// TIA Portal V19 export
FUNCTION "FC30_DoorAcces" : Void   // FC30, LAD
{ S7_Optimized_Access := 'TRUE' }
// stored: AutoNumber false, IsIECCheckEnabled true, SetENOAutomatically false
   VAR_TEMP
      xt_RobotStopped : Bool;
      xt_Robot1Stopped : Bool;
      xt_Robot2Stopped : Bool;
   END_VAR
BEGIN

REGION Network 1: Robot 1 is stopped
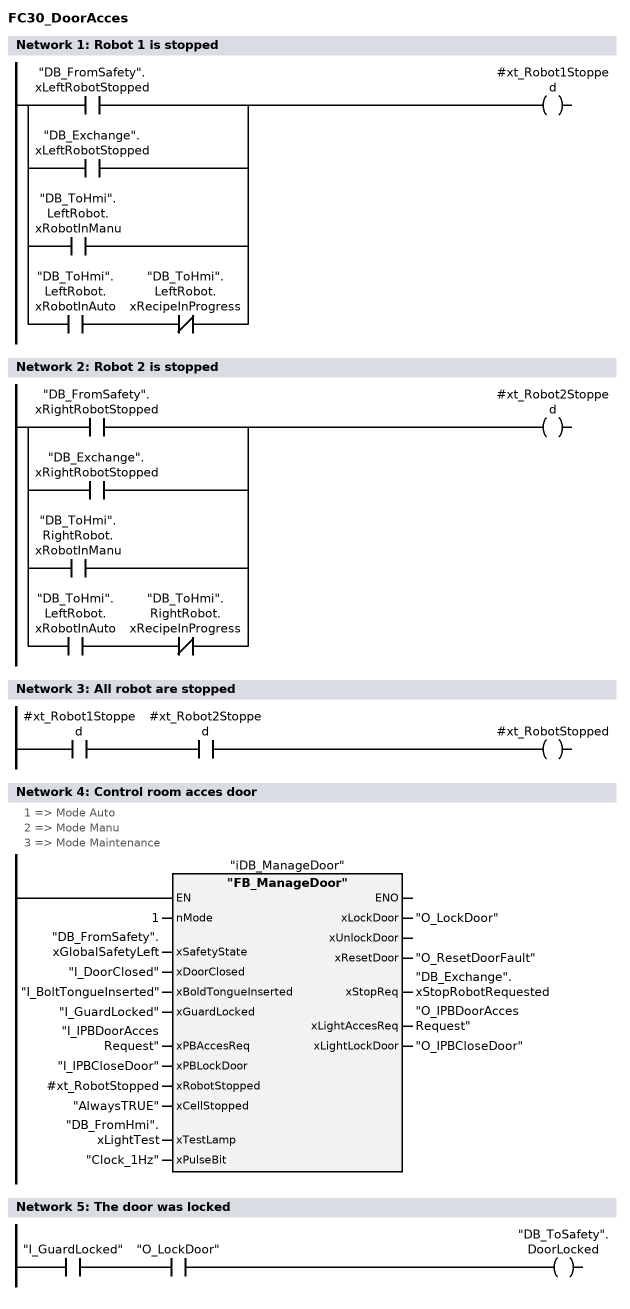
   RUNG wire#powerrail
      Contact( "DB_FromSafety".xLeftRobotStopped )
      wire#w1
      Coil( #xt_Robot1Stopped )
   END_RUNG
   RUNG wire#powerrail
      Contact( "DB_Exchange".xLeftRobotStopped )
   END_RUNG wire#w1
   RUNG wire#powerrail
      Contact( "DB_ToHmi".LeftRobot.xRobotInManu )
   END_RUNG wire#w1
   RUNG wire#powerrail
      Contact( "DB_ToHmi".LeftRobot.xRobotInAuto )
      I_Contact( "DB_ToHmi".LeftRobot.xRecipeInProgress )
   END_RUNG wire#w1
   // the same network as SCL:
   #xt_Robot1Stopped := "DB_FromSafety".xLeftRobotStopped OR "DB_Exchange".xLeftRobotStopped OR "DB_ToHmi".LeftRobot.xRobotInManu OR ("DB_ToHmi".LeftRobot.xRobotInAuto AND NOT "DB_ToHmi".LeftRobot.xRecipeInProgress);
END_REGION

REGION Network 2: Robot 2 is stopped
   RUNG wire#powerrail
      Contact( "DB_FromSafety".xRightRobotStopped )
      wire#w1
      Coil( #xt_Robot2Stopped )
   END_RUNG
   RUNG wire#powerrail
      Contact( "DB_Exchange".xRightRobotStopped )
   END_RUNG wire#w1
   RUNG wire#powerrail
      Contact( "DB_ToHmi".RightRobot.xRobotInManu )
   END_RUNG wire#w1
   RUNG wire#powerrail
      Contact( "DB_ToHmi".LeftRobot.xRobotInAuto )
      I_Contact( "DB_ToHmi".RightRobot.xRecipeInProgress )
   END_RUNG wire#w1
   // the same network as SCL:
   #xt_Robot2Stopped := "DB_FromSafety".xRightRobotStopped OR "DB_Exchange".xRightRobotStopped OR "DB_ToHmi".RightRobot.xRobotInManu OR ("DB_ToHmi".LeftRobot.xRobotInAuto AND NOT "DB_ToHmi".RightRobot.xRecipeInProgress);
END_REGION

REGION Network 3: All robot are stopped
   RUNG wire#powerrail
      Contact( #xt_Robot1Stopped )
      Contact( #xt_Robot2Stopped )
      Coil( #xt_RobotStopped )
   END_RUNG
   // the same network as SCL:
   #xt_RobotStopped := #xt_Robot1Stopped AND #xt_Robot2Stopped;
END_REGION

REGION Network 4: Control room acces door
   // 1 => Mode Auto
   // 2 => Mode Manu
   // 3 => Mode Maintenance
   RUNG wire#powerrail
      "iDB_ManageDoor"(nMode := 1, xSafetyState := "DB_FromSafety".xGlobalSafetyLeft, xDoorClosed := "I_DoorClosed", xBoldTongueInserted := "I_BoltTongueInserted", xGuardLocked := "I_GuardLocked", xPBAccesReq := "I_IPBDoorAccesRequest", xPBLockDoor := "I_IPBCloseDoor", xRobotStopped := #xt_RobotStopped, xCellStopped := "AlwaysTRUE", xTestLamp := "DB_FromHmi".xLightTest, xPulseBit := "Clock_1Hz", xLockDoor => "O_LockDoor", xUnlockDoor =>, xResetDoor => "O_ResetDoorFault", xStopReq => "DB_Exchange".xStopRobotRequested, xLightAccesReq => "O_IPBDoorAccesRequest", xLightLockDoor => "O_IPBCloseDoor")
   END_RUNG
   // the same network as SCL:
   "iDB_ManageDoor"(nMode := 1,   // "FB_ManageDoor"
                    xSafetyState := "DB_FromSafety".xGlobalSafetyLeft,
                    xDoorClosed := "I_DoorClosed",
                    xBoldTongueInserted := "I_BoltTongueInserted",
                    xGuardLocked := "I_GuardLocked",
                    xPBAccesReq := "I_IPBDoorAccesRequest",
                    xPBLockDoor := "I_IPBCloseDoor",
                    xRobotStopped := #xt_RobotStopped,
                    xCellStopped := "AlwaysTRUE",
                    xTestLamp := "DB_FromHmi".xLightTest,
                    xPulseBit := "Clock_1Hz",
                    xLockDoor => "O_LockDoor",
                    xResetDoor => "O_ResetDoorFault",
                    xStopReq => "DB_Exchange".xStopRobotRequested,
                    xLightAccesReq => "O_IPBDoorAccesRequest",
                    xLightLockDoor => "O_IPBCloseDoor");
END_REGION

REGION Network 5: The door was locked
   RUNG wire#powerrail
      Contact( "I_GuardLocked" )
      Contact( "O_LockDoor" )
      Coil( "DB_ToSafety".DoorLocked )
   END_RUNG
   // the same network as SCL:
   "DB_ToSafety".DoorLocked := "I_GuardLocked" AND "O_LockDoor";
END_REGION
END_FUNCTION
